// TIA Portal V17 export
// export: Created 2025-03-07T09:24:06.9571705Z, ExportSetting WithDefaults, DisplayName Totally Integrated Automation Portal, DisplayVersion V17 Update 8, DisplayName TIA Portal Openness, DisplayVersion V17 Update 8, DisplayName TIA Portal Version Control Interface, DisplayVersion V17, DisplayName SINAMICS Startdrive Advanced, DisplayVersion V17 SP2, DisplayName SINAMICS Startdrive G110M, G120, G120C, G120D, G120P, G115D, DisplayVersion V17 SP2, DisplayName SINAMICS Startdrive G130, G150, S120, S150, SINAMICS MV, S210, DisplayVersion V17 SP2, DisplayName STEP 7 Professional, DisplayVersion V17 Update 8, DisplayName SINUMERIK ONE STEP 7 Toolbox, DisplayVersion V17 Update 12, DisplayName SINUMERIK 840D sl STEP 7 Toolbox, DisplayVersion V17 Update 12, DisplayName STEP 7 Safety, DisplayVersion V17 Update 6, DisplayName WinCC Advanced, DisplayVersion V17 Update 8
FUNCTION "FC22701_LOAD_FEEDER_SEQUENCES" : Void   // FC22701, LAD
TITLE = FC22701 LOAD FEEDER SEQUENCES
{ S7_Optimized_Access := 'TRUE' }
VERSION : 0.1
// stored: AutoNumber false, IsIECCheckEnabled false, SetENOAutomatically false, UDAEnableTagReadback false
BEGIN

REGION Network 1: //////////_UNIT_01_//////////
END_REGION

REGION Network 2: /////_HOPPER_1_SEQUENCES_/////
END_REGION

REGION Network 3: CALL FB22701 LOAD FEEDER SEQUENCE TIME UNIT 01 HOPPER 1
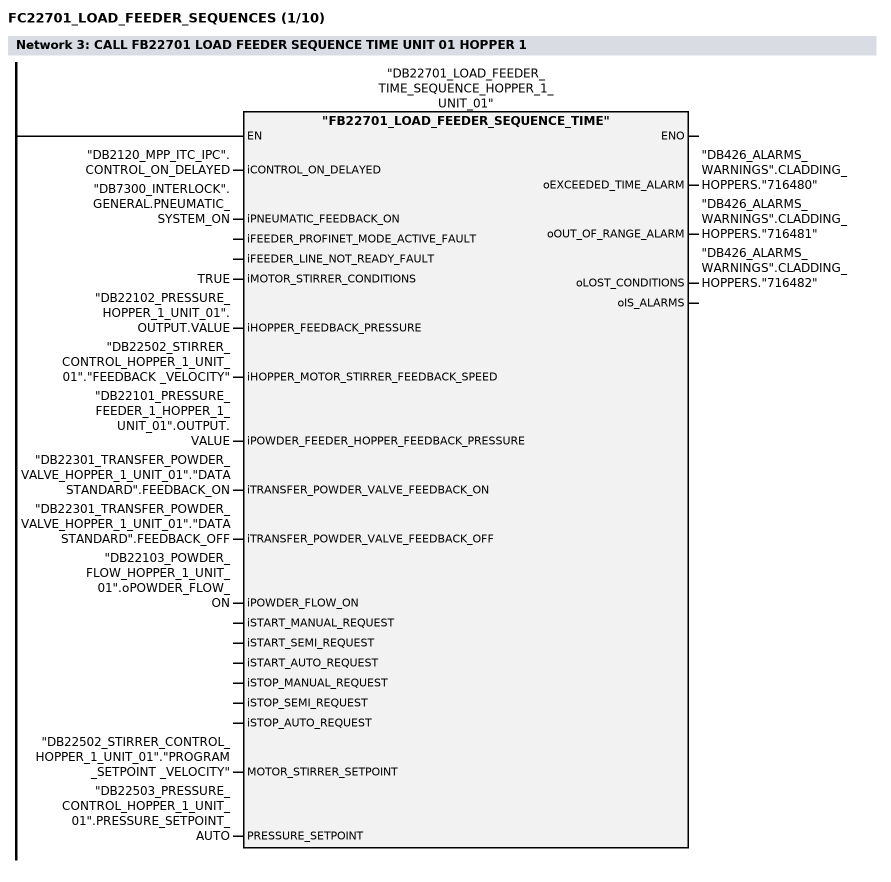
   RUNG wire#powerrail
      "DB22701_LOAD_FEEDER_TIME_SEQUENCE_HOPPER_1_UNIT_01"(iCONTROL_ON_DELAYED := "DB2120_MPP_ITC_IPC".CONTROL_ON_DELAYED, iPNEUMATIC_FEEDBACK_ON := "DB7300_INTERLOCK".GENERAL.PNEUMATIC_SYSTEM_ON, iFEEDER_PROFINET_MODE_ACTIVE_FAULT :=, iFEEDER_LINE_NOT_READY_FAULT :=, iMOTOR_STIRRER_CONDITIONS := TRUE, iHOPPER_FEEDBACK_PRESSURE := "DB22102_PRESSURE_HOPPER_1_UNIT_01".OUTPUT.VALUE, iHOPPER_MOTOR_STIRRER_FEEDBACK_SPEED := "DB22502_STIRRER_CONTROL_HOPPER_1_UNIT_01"."FEEDBACK _VELOCITY", iPOWDER_FEEDER_HOPPER_FEEDBACK_PRESSURE := "DB22101_PRESSURE_FEEDER_1_HOPPER_1_UNIT_01".OUTPUT.VALUE, iTRANSFER_POWDER_VALVE_FEEDBACK_ON := "DB22301_TRANSFER_POWDER_VALVE_HOPPER_1_UNIT_01"."DATA STANDARD".FEEDBACK_ON, iTRANSFER_POWDER_VALVE_FEEDBACK_OFF := "DB22301_TRANSFER_POWDER_VALVE_HOPPER_1_UNIT_01"."DATA STANDARD".FEEDBACK_OFF, iPOWDER_FLOW_ON := "DB22103_POWDER_FLOW_HOPPER_1_UNIT_01".oPOWDER_FLOW_ON, iSTART_MANUAL_REQUEST :=, iSTART_SEMI_REQUEST :=, iSTART_AUTO_REQUEST :=, iSTOP_MANUAL_REQUEST :=, iSTOP_SEMI_REQUEST :=, iSTOP_AUTO_REQUEST :=, MOTOR_STIRRER_SETPOINT := "DB22502_STIRRER_CONTROL_HOPPER_1_UNIT_01"."PROGRAM _SETPOINT _VELOCITY", PRESSURE_SETPOINT := "DB22503_PRESSURE_CONTROL_HOPPER_1_UNIT_01".PRESSURE_SETPOINT_AUTO, oEXCEEDED_TIME_ALARM => "DB426_ALARMS_WARNINGS".CLADDING_HOPPERS."716480", oOUT_OF_RANGE_ALARM => "DB426_ALARMS_WARNINGS".CLADDING_HOPPERS."716481", oLOST_CONDITIONS => "DB426_ALARMS_WARNINGS".CLADDING_HOPPERS."716482", oIS_ALARMS =>)
   END_RUNG
   // the same network as SCL:
   "DB22701_LOAD_FEEDER_TIME_SEQUENCE_HOPPER_1_UNIT_01"(iCONTROL_ON_DELAYED := "DB2120_MPP_ITC_IPC".CONTROL_ON_DELAYED,   // "FB22701_LOAD_FEEDER_SEQUENCE_TIME"
                           iPNEUMATIC_FEEDBACK_ON := "DB7300_INTERLOCK".GENERAL.PNEUMATIC_SYSTEM_ON,
                           iMOTOR_STIRRER_CONDITIONS := TRUE,
                           iHOPPER_FEEDBACK_PRESSURE := "DB22102_PRESSURE_HOPPER_1_UNIT_01".OUTPUT.VALUE,
                           iHOPPER_MOTOR_STIRRER_FEEDBACK_SPEED := "DB22502_STIRRER_CONTROL_HOPPER_1_UNIT_01"."FEEDBACK _VELOCITY",
                           iPOWDER_FEEDER_HOPPER_FEEDBACK_PRESSURE := "DB22101_PRESSURE_FEEDER_1_HOPPER_1_UNIT_01".OUTPUT.VALUE,
                           iTRANSFER_POWDER_VALVE_FEEDBACK_ON := "DB22301_TRANSFER_POWDER_VALVE_HOPPER_1_UNIT_01"."DATA STANDARD".FEEDBACK_ON,
                           iTRANSFER_POWDER_VALVE_FEEDBACK_OFF := "DB22301_TRANSFER_POWDER_VALVE_HOPPER_1_UNIT_01"."DATA STANDARD".FEEDBACK_OFF,
                           iPOWDER_FLOW_ON := "DB22103_POWDER_FLOW_HOPPER_1_UNIT_01".oPOWDER_FLOW_ON,
                           MOTOR_STIRRER_SETPOINT := "DB22502_STIRRER_CONTROL_HOPPER_1_UNIT_01"."PROGRAM _SETPOINT _VELOCITY",
                           PRESSURE_SETPOINT := "DB22503_PRESSURE_CONTROL_HOPPER_1_UNIT_01".PRESSURE_SETPOINT_AUTO,
                           oEXCEEDED_TIME_ALARM => "DB426_ALARMS_WARNINGS".CLADDING_HOPPERS."716480",
                           oOUT_OF_RANGE_ALARM => "DB426_ALARMS_WARNINGS".CLADDING_HOPPERS."716481",
                           oLOST_CONDITIONS => "DB426_ALARMS_WARNINGS".CLADDING_HOPPERS."716482");
END_REGION

REGION Network 4: CALL FB22702 LOAD FEEDER SEQUENCE WEIGHT UNIT 01 HOPPER 1
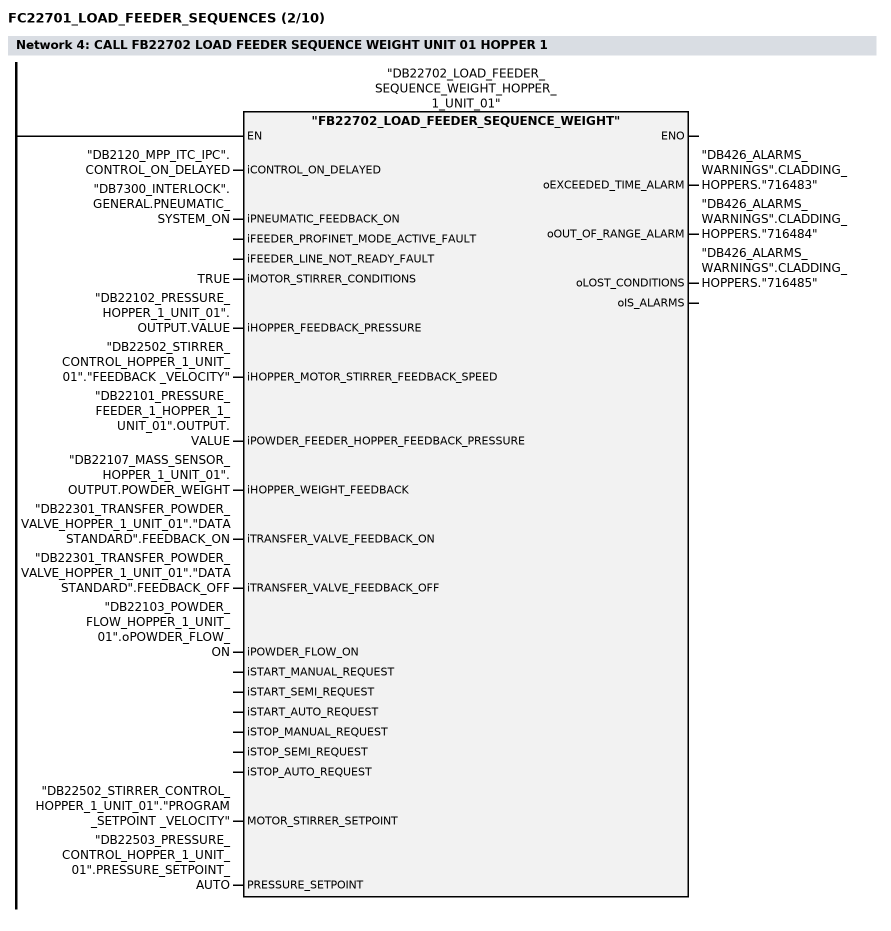
   RUNG wire#powerrail
      "DB22702_LOAD_FEEDER_SEQUENCE_WEIGHT_HOPPER_1_UNIT_01"(iCONTROL_ON_DELAYED := "DB2120_MPP_ITC_IPC".CONTROL_ON_DELAYED, iPNEUMATIC_FEEDBACK_ON := "DB7300_INTERLOCK".GENERAL.PNEUMATIC_SYSTEM_ON, iFEEDER_PROFINET_MODE_ACTIVE_FAULT :=, iFEEDER_LINE_NOT_READY_FAULT :=, iMOTOR_STIRRER_CONDITIONS := TRUE, iHOPPER_FEEDBACK_PRESSURE := "DB22102_PRESSURE_HOPPER_1_UNIT_01".OUTPUT.VALUE, iHOPPER_MOTOR_STIRRER_FEEDBACK_SPEED := "DB22502_STIRRER_CONTROL_HOPPER_1_UNIT_01"."FEEDBACK _VELOCITY", iPOWDER_FEEDER_HOPPER_FEEDBACK_PRESSURE := "DB22101_PRESSURE_FEEDER_1_HOPPER_1_UNIT_01".OUTPUT.VALUE, iHOPPER_WEIGHT_FEEDBACK := "DB22107_MASS_SENSOR_HOPPER_1_UNIT_01".OUTPUT.POWDER_WEIGHT, iTRANSFER_VALVE_FEEDBACK_ON := "DB22301_TRANSFER_POWDER_VALVE_HOPPER_1_UNIT_01"."DATA STANDARD".FEEDBACK_ON, iTRANSFER_VALVE_FEEDBACK_OFF := "DB22301_TRANSFER_POWDER_VALVE_HOPPER_1_UNIT_01"."DATA STANDARD".FEEDBACK_OFF, iPOWDER_FLOW_ON := "DB22103_POWDER_FLOW_HOPPER_1_UNIT_01".oPOWDER_FLOW_ON, iSTART_MANUAL_REQUEST :=, iSTART_SEMI_REQUEST :=, iSTART_AUTO_REQUEST :=, iSTOP_MANUAL_REQUEST :=, iSTOP_SEMI_REQUEST :=, iSTOP_AUTO_REQUEST :=, MOTOR_STIRRER_SETPOINT := "DB22502_STIRRER_CONTROL_HOPPER_1_UNIT_01"."PROGRAM _SETPOINT _VELOCITY", PRESSURE_SETPOINT := "DB22503_PRESSURE_CONTROL_HOPPER_1_UNIT_01".PRESSURE_SETPOINT_AUTO, oEXCEEDED_TIME_ALARM => "DB426_ALARMS_WARNINGS".CLADDING_HOPPERS."716483", oOUT_OF_RANGE_ALARM => "DB426_ALARMS_WARNINGS".CLADDING_HOPPERS."716484", oLOST_CONDITIONS => "DB426_ALARMS_WARNINGS".CLADDING_HOPPERS."716485", oIS_ALARMS =>)
   END_RUNG
   // the same network as SCL:
   "DB22702_LOAD_FEEDER_SEQUENCE_WEIGHT_HOPPER_1_UNIT_01"(iCONTROL_ON_DELAYED := "DB2120_MPP_ITC_IPC".CONTROL_ON_DELAYED,   // "FB22702_LOAD_FEEDER_SEQUENCE_WEIGHT"
                           iPNEUMATIC_FEEDBACK_ON := "DB7300_INTERLOCK".GENERAL.PNEUMATIC_SYSTEM_ON,
                           iMOTOR_STIRRER_CONDITIONS := TRUE,
                           iHOPPER_FEEDBACK_PRESSURE := "DB22102_PRESSURE_HOPPER_1_UNIT_01".OUTPUT.VALUE,
                           iHOPPER_MOTOR_STIRRER_FEEDBACK_SPEED := "DB22502_STIRRER_CONTROL_HOPPER_1_UNIT_01"."FEEDBACK _VELOCITY",
                           iPOWDER_FEEDER_HOPPER_FEEDBACK_PRESSURE := "DB22101_PRESSURE_FEEDER_1_HOPPER_1_UNIT_01".OUTPUT.VALUE,
                           iHOPPER_WEIGHT_FEEDBACK := "DB22107_MASS_SENSOR_HOPPER_1_UNIT_01".OUTPUT.POWDER_WEIGHT,
                           iTRANSFER_VALVE_FEEDBACK_ON := "DB22301_TRANSFER_POWDER_VALVE_HOPPER_1_UNIT_01"."DATA STANDARD".FEEDBACK_ON,
                           iTRANSFER_VALVE_FEEDBACK_OFF := "DB22301_TRANSFER_POWDER_VALVE_HOPPER_1_UNIT_01"."DATA STANDARD".FEEDBACK_OFF,
                           iPOWDER_FLOW_ON := "DB22103_POWDER_FLOW_HOPPER_1_UNIT_01".oPOWDER_FLOW_ON,
                           MOTOR_STIRRER_SETPOINT := "DB22502_STIRRER_CONTROL_HOPPER_1_UNIT_01"."PROGRAM _SETPOINT _VELOCITY",
                           PRESSURE_SETPOINT := "DB22503_PRESSURE_CONTROL_HOPPER_1_UNIT_01".PRESSURE_SETPOINT_AUTO,
                           oEXCEEDED_TIME_ALARM => "DB426_ALARMS_WARNINGS".CLADDING_HOPPERS."716483",
                           oOUT_OF_RANGE_ALARM => "DB426_ALARMS_WARNINGS".CLADDING_HOPPERS."716484",
                           oLOST_CONDITIONS => "DB426_ALARMS_WARNINGS".CLADDING_HOPPERS."716485");
END_REGION

REGION Network 5: /////_HOPPER_2_SEQUENCES_/////
END_REGION

REGION Network 6: CALL FB22701 LOAD FEEDER SEQUENCE TIME UNIT 01 HOPPER 2
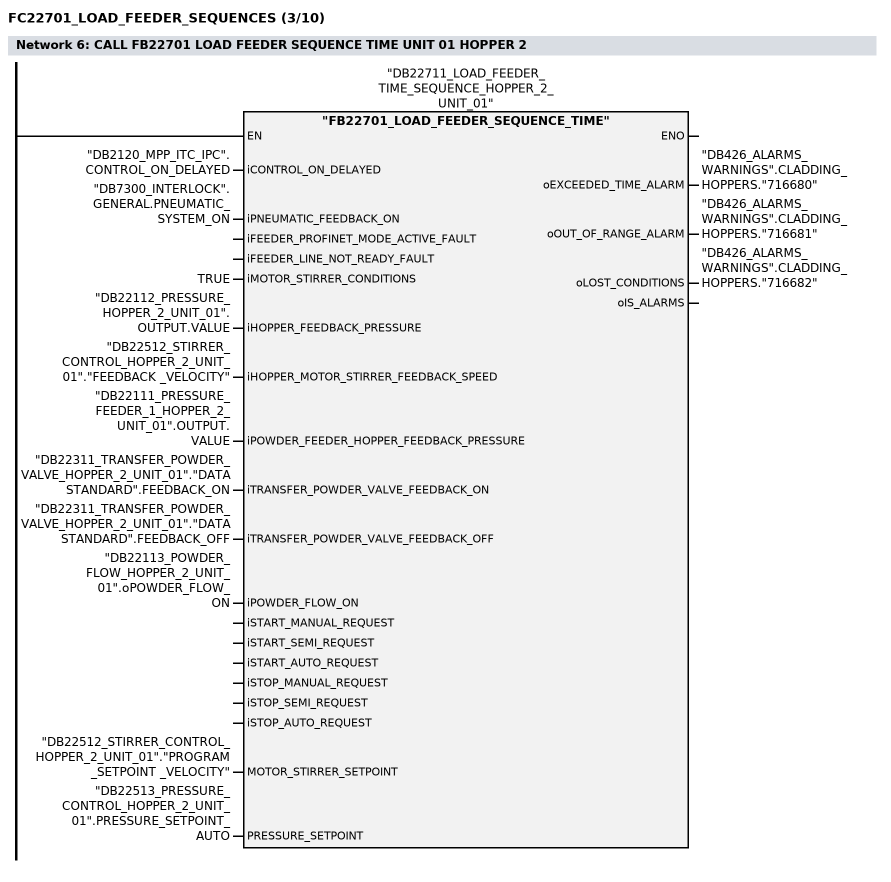
   RUNG wire#powerrail
      "DB22711_LOAD_FEEDER_TIME_SEQUENCE_HOPPER_2_UNIT_01"(iCONTROL_ON_DELAYED := "DB2120_MPP_ITC_IPC".CONTROL_ON_DELAYED, iPNEUMATIC_FEEDBACK_ON := "DB7300_INTERLOCK".GENERAL.PNEUMATIC_SYSTEM_ON, iFEEDER_PROFINET_MODE_ACTIVE_FAULT :=, iFEEDER_LINE_NOT_READY_FAULT :=, iMOTOR_STIRRER_CONDITIONS := TRUE, iHOPPER_FEEDBACK_PRESSURE := "DB22112_PRESSURE_HOPPER_2_UNIT_01".OUTPUT.VALUE, iHOPPER_MOTOR_STIRRER_FEEDBACK_SPEED := "DB22512_STIRRER_CONTROL_HOPPER_2_UNIT_01"."FEEDBACK _VELOCITY", iPOWDER_FEEDER_HOPPER_FEEDBACK_PRESSURE := "DB22111_PRESSURE_FEEDER_1_HOPPER_2_UNIT_01".OUTPUT.VALUE, iTRANSFER_POWDER_VALVE_FEEDBACK_ON := "DB22311_TRANSFER_POWDER_VALVE_HOPPER_2_UNIT_01"."DATA STANDARD".FEEDBACK_ON, iTRANSFER_POWDER_VALVE_FEEDBACK_OFF := "DB22311_TRANSFER_POWDER_VALVE_HOPPER_2_UNIT_01"."DATA STANDARD".FEEDBACK_OFF, iPOWDER_FLOW_ON := "DB22113_POWDER_FLOW_HOPPER_2_UNIT_01".oPOWDER_FLOW_ON, iSTART_MANUAL_REQUEST :=, iSTART_SEMI_REQUEST :=, iSTART_AUTO_REQUEST :=, iSTOP_MANUAL_REQUEST :=, iSTOP_SEMI_REQUEST :=, iSTOP_AUTO_REQUEST :=, MOTOR_STIRRER_SETPOINT := "DB22512_STIRRER_CONTROL_HOPPER_2_UNIT_01"."PROGRAM _SETPOINT _VELOCITY", PRESSURE_SETPOINT := "DB22513_PRESSURE_CONTROL_HOPPER_2_UNIT_01".PRESSURE_SETPOINT_AUTO, oEXCEEDED_TIME_ALARM => "DB426_ALARMS_WARNINGS".CLADDING_HOPPERS."716680", oOUT_OF_RANGE_ALARM => "DB426_ALARMS_WARNINGS".CLADDING_HOPPERS."716681", oLOST_CONDITIONS => "DB426_ALARMS_WARNINGS".CLADDING_HOPPERS."716682", oIS_ALARMS =>)
   END_RUNG
   // the same network as SCL:
   "DB22711_LOAD_FEEDER_TIME_SEQUENCE_HOPPER_2_UNIT_01"(iCONTROL_ON_DELAYED := "DB2120_MPP_ITC_IPC".CONTROL_ON_DELAYED,   // "FB22701_LOAD_FEEDER_SEQUENCE_TIME"
                           iPNEUMATIC_FEEDBACK_ON := "DB7300_INTERLOCK".GENERAL.PNEUMATIC_SYSTEM_ON,
                           iMOTOR_STIRRER_CONDITIONS := TRUE,
                           iHOPPER_FEEDBACK_PRESSURE := "DB22112_PRESSURE_HOPPER_2_UNIT_01".OUTPUT.VALUE,
                           iHOPPER_MOTOR_STIRRER_FEEDBACK_SPEED := "DB22512_STIRRER_CONTROL_HOPPER_2_UNIT_01"."FEEDBACK _VELOCITY",
                           iPOWDER_FEEDER_HOPPER_FEEDBACK_PRESSURE := "DB22111_PRESSURE_FEEDER_1_HOPPER_2_UNIT_01".OUTPUT.VALUE,
                           iTRANSFER_POWDER_VALVE_FEEDBACK_ON := "DB22311_TRANSFER_POWDER_VALVE_HOPPER_2_UNIT_01"."DATA STANDARD".FEEDBACK_ON,
                           iTRANSFER_POWDER_VALVE_FEEDBACK_OFF := "DB22311_TRANSFER_POWDER_VALVE_HOPPER_2_UNIT_01"."DATA STANDARD".FEEDBACK_OFF,
                           iPOWDER_FLOW_ON := "DB22113_POWDER_FLOW_HOPPER_2_UNIT_01".oPOWDER_FLOW_ON,
                           MOTOR_STIRRER_SETPOINT := "DB22512_STIRRER_CONTROL_HOPPER_2_UNIT_01"."PROGRAM _SETPOINT _VELOCITY",
                           PRESSURE_SETPOINT := "DB22513_PRESSURE_CONTROL_HOPPER_2_UNIT_01".PRESSURE_SETPOINT_AUTO,
                           oEXCEEDED_TIME_ALARM => "DB426_ALARMS_WARNINGS".CLADDING_HOPPERS."716680",
                           oOUT_OF_RANGE_ALARM => "DB426_ALARMS_WARNINGS".CLADDING_HOPPERS."716681",
                           oLOST_CONDITIONS => "DB426_ALARMS_WARNINGS".CLADDING_HOPPERS."716682");
END_REGION

REGION Network 7: CALL FB22702 LOAD FEEDER SEQUENCE WEIGHT UNIT 01 HOPPER 2
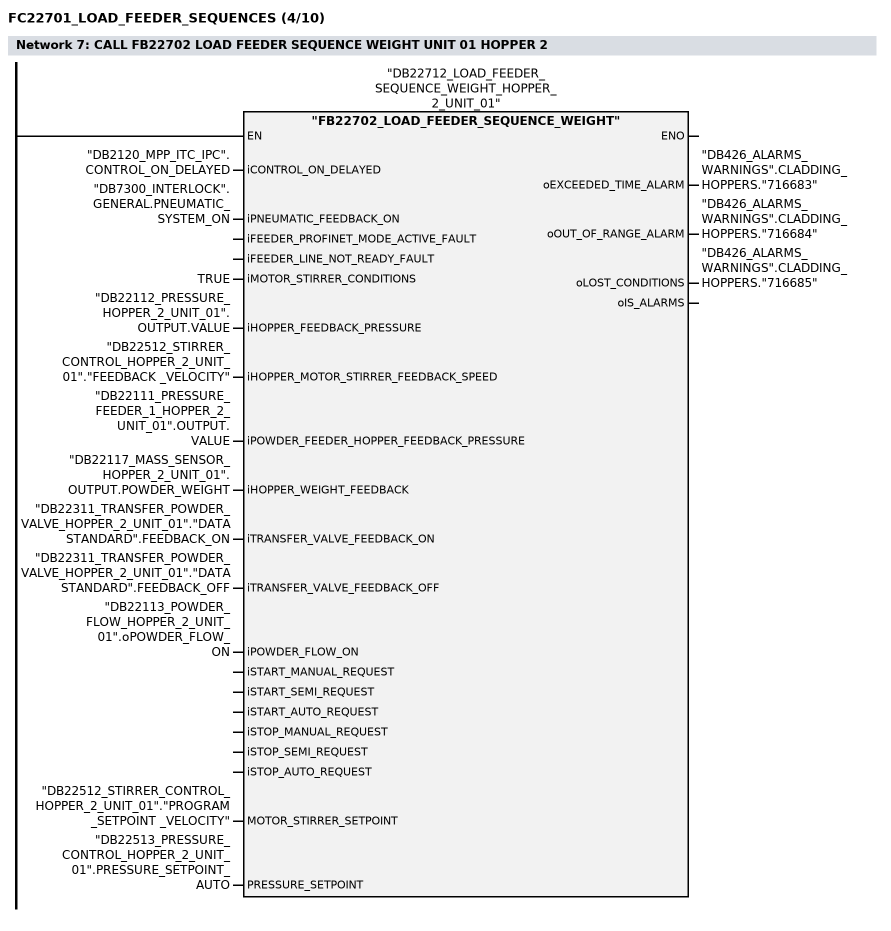
   RUNG wire#powerrail
      "DB22712_LOAD_FEEDER_SEQUENCE_WEIGHT_HOPPER_2_UNIT_01"(iCONTROL_ON_DELAYED := "DB2120_MPP_ITC_IPC".CONTROL_ON_DELAYED, iPNEUMATIC_FEEDBACK_ON := "DB7300_INTERLOCK".GENERAL.PNEUMATIC_SYSTEM_ON, iFEEDER_PROFINET_MODE_ACTIVE_FAULT :=, iFEEDER_LINE_NOT_READY_FAULT :=, iMOTOR_STIRRER_CONDITIONS := TRUE, iHOPPER_FEEDBACK_PRESSURE := "DB22112_PRESSURE_HOPPER_2_UNIT_01".OUTPUT.VALUE, iHOPPER_MOTOR_STIRRER_FEEDBACK_SPEED := "DB22512_STIRRER_CONTROL_HOPPER_2_UNIT_01"."FEEDBACK _VELOCITY", iPOWDER_FEEDER_HOPPER_FEEDBACK_PRESSURE := "DB22111_PRESSURE_FEEDER_1_HOPPER_2_UNIT_01".OUTPUT.VALUE, iHOPPER_WEIGHT_FEEDBACK := "DB22117_MASS_SENSOR_HOPPER_2_UNIT_01".OUTPUT.POWDER_WEIGHT, iTRANSFER_VALVE_FEEDBACK_ON := "DB22311_TRANSFER_POWDER_VALVE_HOPPER_2_UNIT_01"."DATA STANDARD".FEEDBACK_ON, iTRANSFER_VALVE_FEEDBACK_OFF := "DB22311_TRANSFER_POWDER_VALVE_HOPPER_2_UNIT_01"."DATA STANDARD".FEEDBACK_OFF, iPOWDER_FLOW_ON := "DB22113_POWDER_FLOW_HOPPER_2_UNIT_01".oPOWDER_FLOW_ON, iSTART_MANUAL_REQUEST :=, iSTART_SEMI_REQUEST :=, iSTART_AUTO_REQUEST :=, iSTOP_MANUAL_REQUEST :=, iSTOP_SEMI_REQUEST :=, iSTOP_AUTO_REQUEST :=, MOTOR_STIRRER_SETPOINT := "DB22512_STIRRER_CONTROL_HOPPER_2_UNIT_01"."PROGRAM _SETPOINT _VELOCITY", PRESSURE_SETPOINT := "DB22513_PRESSURE_CONTROL_HOPPER_2_UNIT_01".PRESSURE_SETPOINT_AUTO, oEXCEEDED_TIME_ALARM => "DB426_ALARMS_WARNINGS".CLADDING_HOPPERS."716683", oOUT_OF_RANGE_ALARM => "DB426_ALARMS_WARNINGS".CLADDING_HOPPERS."716684", oLOST_CONDITIONS => "DB426_ALARMS_WARNINGS".CLADDING_HOPPERS."716685", oIS_ALARMS =>)
   END_RUNG
   // the same network as SCL:
   "DB22712_LOAD_FEEDER_SEQUENCE_WEIGHT_HOPPER_2_UNIT_01"(iCONTROL_ON_DELAYED := "DB2120_MPP_ITC_IPC".CONTROL_ON_DELAYED,   // "FB22702_LOAD_FEEDER_SEQUENCE_WEIGHT"
                           iPNEUMATIC_FEEDBACK_ON := "DB7300_INTERLOCK".GENERAL.PNEUMATIC_SYSTEM_ON,
                           iMOTOR_STIRRER_CONDITIONS := TRUE,
                           iHOPPER_FEEDBACK_PRESSURE := "DB22112_PRESSURE_HOPPER_2_UNIT_01".OUTPUT.VALUE,
                           iHOPPER_MOTOR_STIRRER_FEEDBACK_SPEED := "DB22512_STIRRER_CONTROL_HOPPER_2_UNIT_01"."FEEDBACK _VELOCITY",
                           iPOWDER_FEEDER_HOPPER_FEEDBACK_PRESSURE := "DB22111_PRESSURE_FEEDER_1_HOPPER_2_UNIT_01".OUTPUT.VALUE,
                           iHOPPER_WEIGHT_FEEDBACK := "DB22117_MASS_SENSOR_HOPPER_2_UNIT_01".OUTPUT.POWDER_WEIGHT,
                           iTRANSFER_VALVE_FEEDBACK_ON := "DB22311_TRANSFER_POWDER_VALVE_HOPPER_2_UNIT_01"."DATA STANDARD".FEEDBACK_ON,
                           iTRANSFER_VALVE_FEEDBACK_OFF := "DB22311_TRANSFER_POWDER_VALVE_HOPPER_2_UNIT_01"."DATA STANDARD".FEEDBACK_OFF,
                           iPOWDER_FLOW_ON := "DB22113_POWDER_FLOW_HOPPER_2_UNIT_01".oPOWDER_FLOW_ON,
                           MOTOR_STIRRER_SETPOINT := "DB22512_STIRRER_CONTROL_HOPPER_2_UNIT_01"."PROGRAM _SETPOINT _VELOCITY",
                           PRESSURE_SETPOINT := "DB22513_PRESSURE_CONTROL_HOPPER_2_UNIT_01".PRESSURE_SETPOINT_AUTO,
                           oEXCEEDED_TIME_ALARM => "DB426_ALARMS_WARNINGS".CLADDING_HOPPERS."716683",
                           oOUT_OF_RANGE_ALARM => "DB426_ALARMS_WARNINGS".CLADDING_HOPPERS."716684",
                           oLOST_CONDITIONS => "DB426_ALARMS_WARNINGS".CLADDING_HOPPERS."716685");
END_REGION

REGION Network 8: //////////_UNIT_02_//////////
END_REGION

REGION Network 9: /////_HOPPER_1_SEQUENCES_/////
END_REGION

REGION Network 10: CALL FB22701 LOAD FEEDER SEQUENCE TIME UNIT 02 HOPPER 1
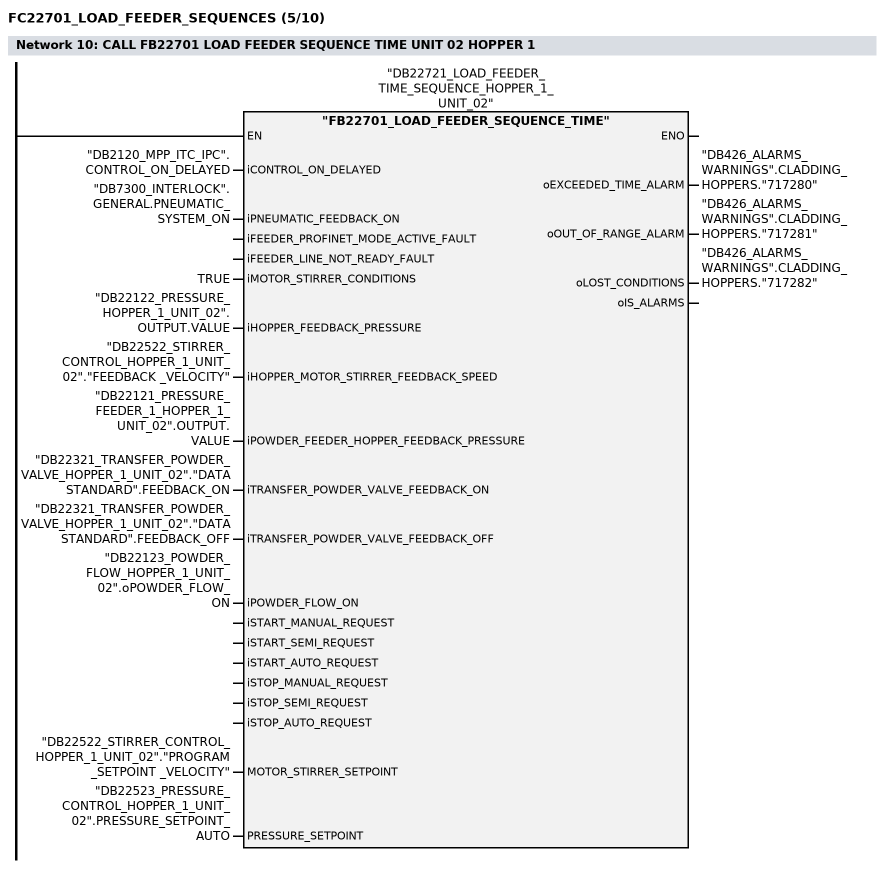
   RUNG wire#powerrail
      "DB22721_LOAD_FEEDER_TIME_SEQUENCE_HOPPER_1_UNIT_02"(iCONTROL_ON_DELAYED := "DB2120_MPP_ITC_IPC".CONTROL_ON_DELAYED, iPNEUMATIC_FEEDBACK_ON := "DB7300_INTERLOCK".GENERAL.PNEUMATIC_SYSTEM_ON, iFEEDER_PROFINET_MODE_ACTIVE_FAULT :=, iFEEDER_LINE_NOT_READY_FAULT :=, iMOTOR_STIRRER_CONDITIONS := TRUE, iHOPPER_FEEDBACK_PRESSURE := "DB22122_PRESSURE_HOPPER_1_UNIT_02".OUTPUT.VALUE, iHOPPER_MOTOR_STIRRER_FEEDBACK_SPEED := "DB22522_STIRRER_CONTROL_HOPPER_1_UNIT_02"."FEEDBACK _VELOCITY", iPOWDER_FEEDER_HOPPER_FEEDBACK_PRESSURE := "DB22121_PRESSURE_FEEDER_1_HOPPER_1_UNIT_02".OUTPUT.VALUE, iTRANSFER_POWDER_VALVE_FEEDBACK_ON := "DB22321_TRANSFER_POWDER_VALVE_HOPPER_1_UNIT_02"."DATA STANDARD".FEEDBACK_ON, iTRANSFER_POWDER_VALVE_FEEDBACK_OFF := "DB22321_TRANSFER_POWDER_VALVE_HOPPER_1_UNIT_02"."DATA STANDARD".FEEDBACK_OFF, iPOWDER_FLOW_ON := "DB22123_POWDER_FLOW_HOPPER_1_UNIT_02".oPOWDER_FLOW_ON, iSTART_MANUAL_REQUEST :=, iSTART_SEMI_REQUEST :=, iSTART_AUTO_REQUEST :=, iSTOP_MANUAL_REQUEST :=, iSTOP_SEMI_REQUEST :=, iSTOP_AUTO_REQUEST :=, MOTOR_STIRRER_SETPOINT := "DB22522_STIRRER_CONTROL_HOPPER_1_UNIT_02"."PROGRAM _SETPOINT _VELOCITY", PRESSURE_SETPOINT := "DB22523_PRESSURE_CONTROL_HOPPER_1_UNIT_02".PRESSURE_SETPOINT_AUTO, oEXCEEDED_TIME_ALARM => "DB426_ALARMS_WARNINGS".CLADDING_HOPPERS."717280", oOUT_OF_RANGE_ALARM => "DB426_ALARMS_WARNINGS".CLADDING_HOPPERS."717281", oLOST_CONDITIONS => "DB426_ALARMS_WARNINGS".CLADDING_HOPPERS."717282", oIS_ALARMS =>)
   END_RUNG
   // the same network as SCL:
   "DB22721_LOAD_FEEDER_TIME_SEQUENCE_HOPPER_1_UNIT_02"(iCONTROL_ON_DELAYED := "DB2120_MPP_ITC_IPC".CONTROL_ON_DELAYED,   // "FB22701_LOAD_FEEDER_SEQUENCE_TIME"
                           iPNEUMATIC_FEEDBACK_ON := "DB7300_INTERLOCK".GENERAL.PNEUMATIC_SYSTEM_ON,
                           iMOTOR_STIRRER_CONDITIONS := TRUE,
                           iHOPPER_FEEDBACK_PRESSURE := "DB22122_PRESSURE_HOPPER_1_UNIT_02".OUTPUT.VALUE,
                           iHOPPER_MOTOR_STIRRER_FEEDBACK_SPEED := "DB22522_STIRRER_CONTROL_HOPPER_1_UNIT_02"."FEEDBACK _VELOCITY",
                           iPOWDER_FEEDER_HOPPER_FEEDBACK_PRESSURE := "DB22121_PRESSURE_FEEDER_1_HOPPER_1_UNIT_02".OUTPUT.VALUE,
                           iTRANSFER_POWDER_VALVE_FEEDBACK_ON := "DB22321_TRANSFER_POWDER_VALVE_HOPPER_1_UNIT_02"."DATA STANDARD".FEEDBACK_ON,
                           iTRANSFER_POWDER_VALVE_FEEDBACK_OFF := "DB22321_TRANSFER_POWDER_VALVE_HOPPER_1_UNIT_02"."DATA STANDARD".FEEDBACK_OFF,
                           iPOWDER_FLOW_ON := "DB22123_POWDER_FLOW_HOPPER_1_UNIT_02".oPOWDER_FLOW_ON,
                           MOTOR_STIRRER_SETPOINT := "DB22522_STIRRER_CONTROL_HOPPER_1_UNIT_02"."PROGRAM _SETPOINT _VELOCITY",
                           PRESSURE_SETPOINT := "DB22523_PRESSURE_CONTROL_HOPPER_1_UNIT_02".PRESSURE_SETPOINT_AUTO,
                           oEXCEEDED_TIME_ALARM => "DB426_ALARMS_WARNINGS".CLADDING_HOPPERS."717280",
                           oOUT_OF_RANGE_ALARM => "DB426_ALARMS_WARNINGS".CLADDING_HOPPERS."717281",
                           oLOST_CONDITIONS => "DB426_ALARMS_WARNINGS".CLADDING_HOPPERS."717282");
END_REGION

REGION Network 11: CALL FB22702 LOAD FEEDER SEQUENCE WEIGHT UNIT 02 HOPPER 1
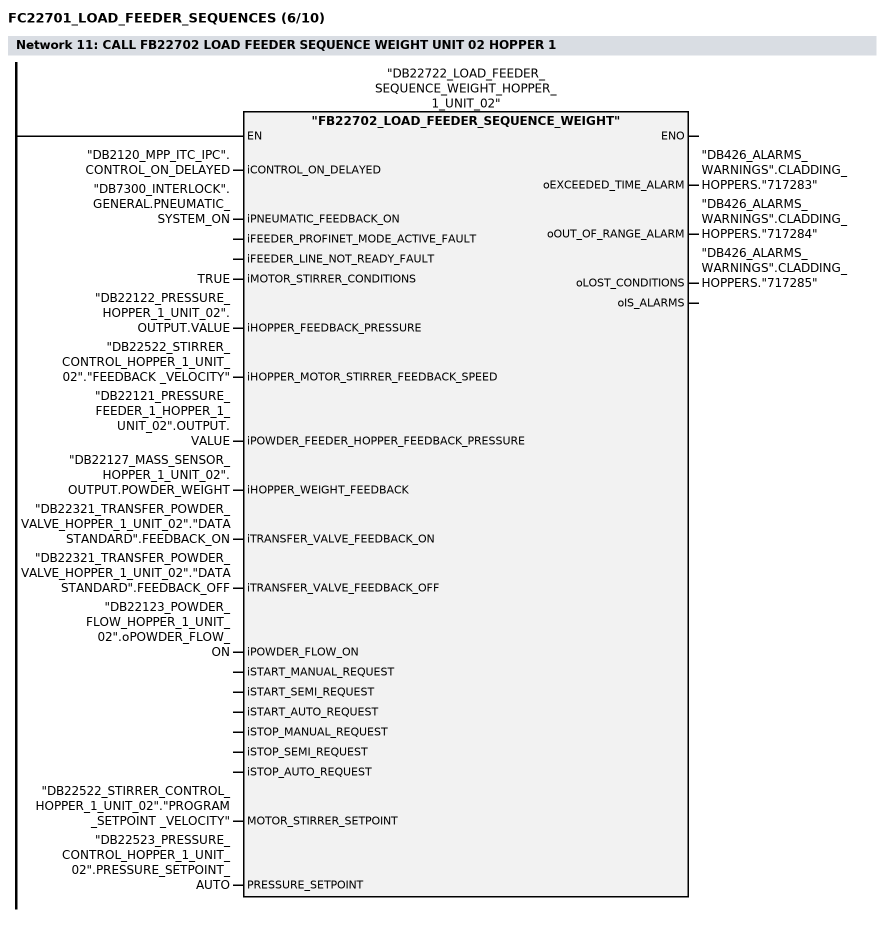
   RUNG wire#powerrail
      "DB22722_LOAD_FEEDER_SEQUENCE_WEIGHT_HOPPER_1_UNIT_02"(iCONTROL_ON_DELAYED := "DB2120_MPP_ITC_IPC".CONTROL_ON_DELAYED, iPNEUMATIC_FEEDBACK_ON := "DB7300_INTERLOCK".GENERAL.PNEUMATIC_SYSTEM_ON, iFEEDER_PROFINET_MODE_ACTIVE_FAULT :=, iFEEDER_LINE_NOT_READY_FAULT :=, iMOTOR_STIRRER_CONDITIONS := TRUE, iHOPPER_FEEDBACK_PRESSURE := "DB22122_PRESSURE_HOPPER_1_UNIT_02".OUTPUT.VALUE, iHOPPER_MOTOR_STIRRER_FEEDBACK_SPEED := "DB22522_STIRRER_CONTROL_HOPPER_1_UNIT_02"."FEEDBACK _VELOCITY", iPOWDER_FEEDER_HOPPER_FEEDBACK_PRESSURE := "DB22121_PRESSURE_FEEDER_1_HOPPER_1_UNIT_02".OUTPUT.VALUE, iHOPPER_WEIGHT_FEEDBACK := "DB22127_MASS_SENSOR_HOPPER_1_UNIT_02".OUTPUT.POWDER_WEIGHT, iTRANSFER_VALVE_FEEDBACK_ON := "DB22321_TRANSFER_POWDER_VALVE_HOPPER_1_UNIT_02"."DATA STANDARD".FEEDBACK_ON, iTRANSFER_VALVE_FEEDBACK_OFF := "DB22321_TRANSFER_POWDER_VALVE_HOPPER_1_UNIT_02"."DATA STANDARD".FEEDBACK_OFF, iPOWDER_FLOW_ON := "DB22123_POWDER_FLOW_HOPPER_1_UNIT_02".oPOWDER_FLOW_ON, iSTART_MANUAL_REQUEST :=, iSTART_SEMI_REQUEST :=, iSTART_AUTO_REQUEST :=, iSTOP_MANUAL_REQUEST :=, iSTOP_SEMI_REQUEST :=, iSTOP_AUTO_REQUEST :=, MOTOR_STIRRER_SETPOINT := "DB22522_STIRRER_CONTROL_HOPPER_1_UNIT_02"."PROGRAM _SETPOINT _VELOCITY", PRESSURE_SETPOINT := "DB22523_PRESSURE_CONTROL_HOPPER_1_UNIT_02".PRESSURE_SETPOINT_AUTO, oEXCEEDED_TIME_ALARM => "DB426_ALARMS_WARNINGS".CLADDING_HOPPERS."717283", oOUT_OF_RANGE_ALARM => "DB426_ALARMS_WARNINGS".CLADDING_HOPPERS."717284", oLOST_CONDITIONS => "DB426_ALARMS_WARNINGS".CLADDING_HOPPERS."717285", oIS_ALARMS =>)
   END_RUNG
   // the same network as SCL:
   "DB22722_LOAD_FEEDER_SEQUENCE_WEIGHT_HOPPER_1_UNIT_02"(iCONTROL_ON_DELAYED := "DB2120_MPP_ITC_IPC".CONTROL_ON_DELAYED,   // "FB22702_LOAD_FEEDER_SEQUENCE_WEIGHT"
                           iPNEUMATIC_FEEDBACK_ON := "DB7300_INTERLOCK".GENERAL.PNEUMATIC_SYSTEM_ON,
                           iMOTOR_STIRRER_CONDITIONS := TRUE,
                           iHOPPER_FEEDBACK_PRESSURE := "DB22122_PRESSURE_HOPPER_1_UNIT_02".OUTPUT.VALUE,
                           iHOPPER_MOTOR_STIRRER_FEEDBACK_SPEED := "DB22522_STIRRER_CONTROL_HOPPER_1_UNIT_02"."FEEDBACK _VELOCITY",
                           iPOWDER_FEEDER_HOPPER_FEEDBACK_PRESSURE := "DB22121_PRESSURE_FEEDER_1_HOPPER_1_UNIT_02".OUTPUT.VALUE,
                           iHOPPER_WEIGHT_FEEDBACK := "DB22127_MASS_SENSOR_HOPPER_1_UNIT_02".OUTPUT.POWDER_WEIGHT,
                           iTRANSFER_VALVE_FEEDBACK_ON := "DB22321_TRANSFER_POWDER_VALVE_HOPPER_1_UNIT_02"."DATA STANDARD".FEEDBACK_ON,
                           iTRANSFER_VALVE_FEEDBACK_OFF := "DB22321_TRANSFER_POWDER_VALVE_HOPPER_1_UNIT_02"."DATA STANDARD".FEEDBACK_OFF,
                           iPOWDER_FLOW_ON := "DB22123_POWDER_FLOW_HOPPER_1_UNIT_02".oPOWDER_FLOW_ON,
                           MOTOR_STIRRER_SETPOINT := "DB22522_STIRRER_CONTROL_HOPPER_1_UNIT_02"."PROGRAM _SETPOINT _VELOCITY",
                           PRESSURE_SETPOINT := "DB22523_PRESSURE_CONTROL_HOPPER_1_UNIT_02".PRESSURE_SETPOINT_AUTO,
                           oEXCEEDED_TIME_ALARM => "DB426_ALARMS_WARNINGS".CLADDING_HOPPERS."717283",
                           oOUT_OF_RANGE_ALARM => "DB426_ALARMS_WARNINGS".CLADDING_HOPPERS."717284",
                           oLOST_CONDITIONS => "DB426_ALARMS_WARNINGS".CLADDING_HOPPERS."717285");
END_REGION

REGION Network 12: /////_HOPPER_2_SEQUENCES_/////
END_REGION

REGION Network 13: CALL FB22701 LOAD FEEDER SEQUENCE TIME UNIT 02 HOPPER 2
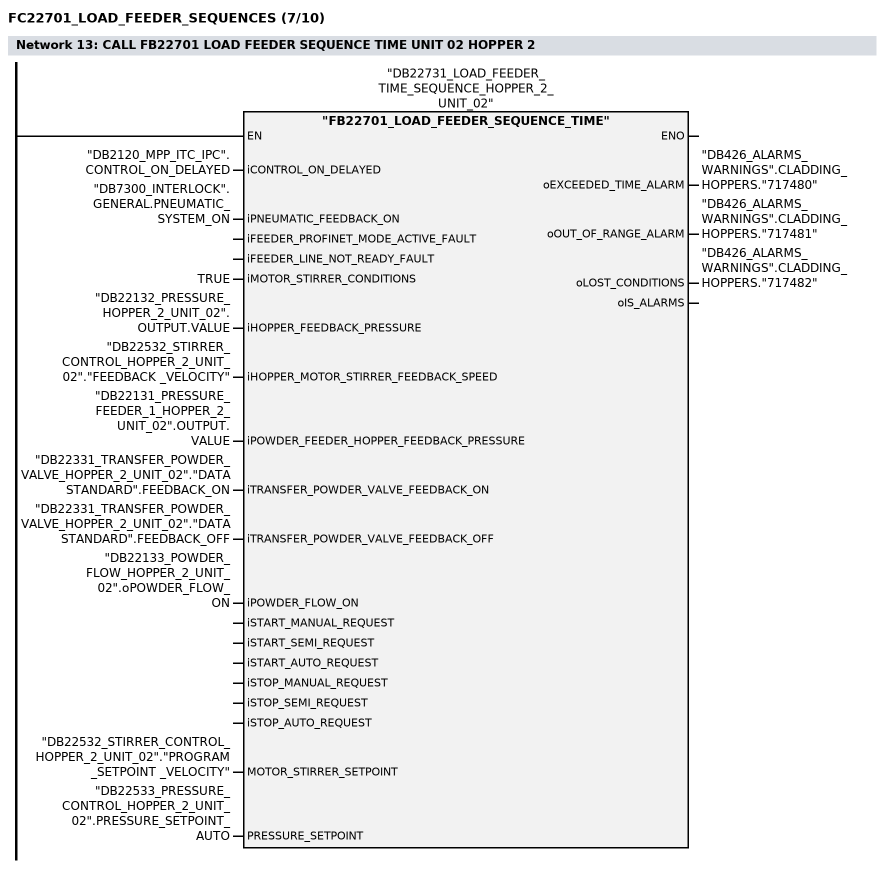
   RUNG wire#powerrail
      "DB22731_LOAD_FEEDER_TIME_SEQUENCE_HOPPER_2_UNIT_02"(iCONTROL_ON_DELAYED := "DB2120_MPP_ITC_IPC".CONTROL_ON_DELAYED, iPNEUMATIC_FEEDBACK_ON := "DB7300_INTERLOCK".GENERAL.PNEUMATIC_SYSTEM_ON, iFEEDER_PROFINET_MODE_ACTIVE_FAULT :=, iFEEDER_LINE_NOT_READY_FAULT :=, iMOTOR_STIRRER_CONDITIONS := TRUE, iHOPPER_FEEDBACK_PRESSURE := "DB22132_PRESSURE_HOPPER_2_UNIT_02".OUTPUT.VALUE, iHOPPER_MOTOR_STIRRER_FEEDBACK_SPEED := "DB22532_STIRRER_CONTROL_HOPPER_2_UNIT_02"."FEEDBACK _VELOCITY", iPOWDER_FEEDER_HOPPER_FEEDBACK_PRESSURE := "DB22131_PRESSURE_FEEDER_1_HOPPER_2_UNIT_02".OUTPUT.VALUE, iTRANSFER_POWDER_VALVE_FEEDBACK_ON := "DB22331_TRANSFER_POWDER_VALVE_HOPPER_2_UNIT_02"."DATA STANDARD".FEEDBACK_ON, iTRANSFER_POWDER_VALVE_FEEDBACK_OFF := "DB22331_TRANSFER_POWDER_VALVE_HOPPER_2_UNIT_02"."DATA STANDARD".FEEDBACK_OFF, iPOWDER_FLOW_ON := "DB22133_POWDER_FLOW_HOPPER_2_UNIT_02".oPOWDER_FLOW_ON, iSTART_MANUAL_REQUEST :=, iSTART_SEMI_REQUEST :=, iSTART_AUTO_REQUEST :=, iSTOP_MANUAL_REQUEST :=, iSTOP_SEMI_REQUEST :=, iSTOP_AUTO_REQUEST :=, MOTOR_STIRRER_SETPOINT := "DB22532_STIRRER_CONTROL_HOPPER_2_UNIT_02"."PROGRAM _SETPOINT _VELOCITY", PRESSURE_SETPOINT := "DB22533_PRESSURE_CONTROL_HOPPER_2_UNIT_02".PRESSURE_SETPOINT_AUTO, oEXCEEDED_TIME_ALARM => "DB426_ALARMS_WARNINGS".CLADDING_HOPPERS."717480", oOUT_OF_RANGE_ALARM => "DB426_ALARMS_WARNINGS".CLADDING_HOPPERS."717481", oLOST_CONDITIONS => "DB426_ALARMS_WARNINGS".CLADDING_HOPPERS."717482", oIS_ALARMS =>)
   END_RUNG
   // the same network as SCL:
   "DB22731_LOAD_FEEDER_TIME_SEQUENCE_HOPPER_2_UNIT_02"(iCONTROL_ON_DELAYED := "DB2120_MPP_ITC_IPC".CONTROL_ON_DELAYED,   // "FB22701_LOAD_FEEDER_SEQUENCE_TIME"
                           iPNEUMATIC_FEEDBACK_ON := "DB7300_INTERLOCK".GENERAL.PNEUMATIC_SYSTEM_ON,
                           iMOTOR_STIRRER_CONDITIONS := TRUE,
                           iHOPPER_FEEDBACK_PRESSURE := "DB22132_PRESSURE_HOPPER_2_UNIT_02".OUTPUT.VALUE,
                           iHOPPER_MOTOR_STIRRER_FEEDBACK_SPEED := "DB22532_STIRRER_CONTROL_HOPPER_2_UNIT_02"."FEEDBACK _VELOCITY",
                           iPOWDER_FEEDER_HOPPER_FEEDBACK_PRESSURE := "DB22131_PRESSURE_FEEDER_1_HOPPER_2_UNIT_02".OUTPUT.VALUE,
                           iTRANSFER_POWDER_VALVE_FEEDBACK_ON := "DB22331_TRANSFER_POWDER_VALVE_HOPPER_2_UNIT_02"."DATA STANDARD".FEEDBACK_ON,
                           iTRANSFER_POWDER_VALVE_FEEDBACK_OFF := "DB22331_TRANSFER_POWDER_VALVE_HOPPER_2_UNIT_02"."DATA STANDARD".FEEDBACK_OFF,
                           iPOWDER_FLOW_ON := "DB22133_POWDER_FLOW_HOPPER_2_UNIT_02".oPOWDER_FLOW_ON,
                           MOTOR_STIRRER_SETPOINT := "DB22532_STIRRER_CONTROL_HOPPER_2_UNIT_02"."PROGRAM _SETPOINT _VELOCITY",
                           PRESSURE_SETPOINT := "DB22533_PRESSURE_CONTROL_HOPPER_2_UNIT_02".PRESSURE_SETPOINT_AUTO,
                           oEXCEEDED_TIME_ALARM => "DB426_ALARMS_WARNINGS".CLADDING_HOPPERS."717480",
                           oOUT_OF_RANGE_ALARM => "DB426_ALARMS_WARNINGS".CLADDING_HOPPERS."717481",
                           oLOST_CONDITIONS => "DB426_ALARMS_WARNINGS".CLADDING_HOPPERS."717482");
END_REGION

REGION Network 14: CALL FB22702 LOAD FEEDER SEQUENCE WEIGHT UNIT 02 HOPPER 2
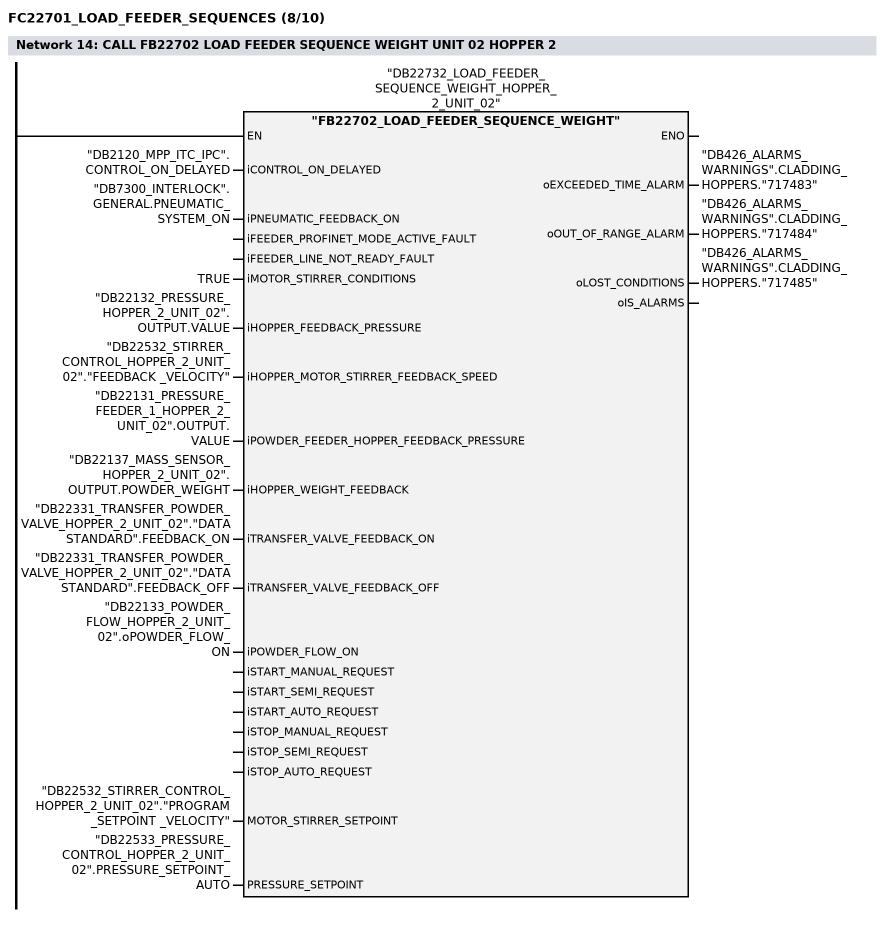
   RUNG wire#powerrail
      "DB22732_LOAD_FEEDER_SEQUENCE_WEIGHT_HOPPER_2_UNIT_02"(iCONTROL_ON_DELAYED := "DB2120_MPP_ITC_IPC".CONTROL_ON_DELAYED, iPNEUMATIC_FEEDBACK_ON := "DB7300_INTERLOCK".GENERAL.PNEUMATIC_SYSTEM_ON, iFEEDER_PROFINET_MODE_ACTIVE_FAULT :=, iFEEDER_LINE_NOT_READY_FAULT :=, iMOTOR_STIRRER_CONDITIONS := TRUE, iHOPPER_FEEDBACK_PRESSURE := "DB22132_PRESSURE_HOPPER_2_UNIT_02".OUTPUT.VALUE, iHOPPER_MOTOR_STIRRER_FEEDBACK_SPEED := "DB22532_STIRRER_CONTROL_HOPPER_2_UNIT_02"."FEEDBACK _VELOCITY", iPOWDER_FEEDER_HOPPER_FEEDBACK_PRESSURE := "DB22131_PRESSURE_FEEDER_1_HOPPER_2_UNIT_02".OUTPUT.VALUE, iHOPPER_WEIGHT_FEEDBACK := "DB22137_MASS_SENSOR_HOPPER_2_UNIT_02".OUTPUT.POWDER_WEIGHT, iTRANSFER_VALVE_FEEDBACK_ON := "DB22331_TRANSFER_POWDER_VALVE_HOPPER_2_UNIT_02"."DATA STANDARD".FEEDBACK_ON, iTRANSFER_VALVE_FEEDBACK_OFF := "DB22331_TRANSFER_POWDER_VALVE_HOPPER_2_UNIT_02"."DATA STANDARD".FEEDBACK_OFF, iPOWDER_FLOW_ON := "DB22133_POWDER_FLOW_HOPPER_2_UNIT_02".oPOWDER_FLOW_ON, iSTART_MANUAL_REQUEST :=, iSTART_SEMI_REQUEST :=, iSTART_AUTO_REQUEST :=, iSTOP_MANUAL_REQUEST :=, iSTOP_SEMI_REQUEST :=, iSTOP_AUTO_REQUEST :=, MOTOR_STIRRER_SETPOINT := "DB22532_STIRRER_CONTROL_HOPPER_2_UNIT_02"."PROGRAM _SETPOINT _VELOCITY", PRESSURE_SETPOINT := "DB22533_PRESSURE_CONTROL_HOPPER_2_UNIT_02".PRESSURE_SETPOINT_AUTO, oEXCEEDED_TIME_ALARM => "DB426_ALARMS_WARNINGS".CLADDING_HOPPERS."717483", oOUT_OF_RANGE_ALARM => "DB426_ALARMS_WARNINGS".CLADDING_HOPPERS."717484", oLOST_CONDITIONS => "DB426_ALARMS_WARNINGS".CLADDING_HOPPERS."717485", oIS_ALARMS =>)
   END_RUNG
   // the same network as SCL:
   "DB22732_LOAD_FEEDER_SEQUENCE_WEIGHT_HOPPER_2_UNIT_02"(iCONTROL_ON_DELAYED := "DB2120_MPP_ITC_IPC".CONTROL_ON_DELAYED,   // "FB22702_LOAD_FEEDER_SEQUENCE_WEIGHT"
                           iPNEUMATIC_FEEDBACK_ON := "DB7300_INTERLOCK".GENERAL.PNEUMATIC_SYSTEM_ON,
                           iMOTOR_STIRRER_CONDITIONS := TRUE,
                           iHOPPER_FEEDBACK_PRESSURE := "DB22132_PRESSURE_HOPPER_2_UNIT_02".OUTPUT.VALUE,
                           iHOPPER_MOTOR_STIRRER_FEEDBACK_SPEED := "DB22532_STIRRER_CONTROL_HOPPER_2_UNIT_02"."FEEDBACK _VELOCITY",
                           iPOWDER_FEEDER_HOPPER_FEEDBACK_PRESSURE := "DB22131_PRESSURE_FEEDER_1_HOPPER_2_UNIT_02".OUTPUT.VALUE,
                           iHOPPER_WEIGHT_FEEDBACK := "DB22137_MASS_SENSOR_HOPPER_2_UNIT_02".OUTPUT.POWDER_WEIGHT,
                           iTRANSFER_VALVE_FEEDBACK_ON := "DB22331_TRANSFER_POWDER_VALVE_HOPPER_2_UNIT_02"."DATA STANDARD".FEEDBACK_ON,
                           iTRANSFER_VALVE_FEEDBACK_OFF := "DB22331_TRANSFER_POWDER_VALVE_HOPPER_2_UNIT_02"."DATA STANDARD".FEEDBACK_OFF,
                           iPOWDER_FLOW_ON := "DB22133_POWDER_FLOW_HOPPER_2_UNIT_02".oPOWDER_FLOW_ON,
                           MOTOR_STIRRER_SETPOINT := "DB22532_STIRRER_CONTROL_HOPPER_2_UNIT_02"."PROGRAM _SETPOINT _VELOCITY",
                           PRESSURE_SETPOINT := "DB22533_PRESSURE_CONTROL_HOPPER_2_UNIT_02".PRESSURE_SETPOINT_AUTO,
                           oEXCEEDED_TIME_ALARM => "DB426_ALARMS_WARNINGS".CLADDING_HOPPERS."717483",
                           oOUT_OF_RANGE_ALARM => "DB426_ALARMS_WARNINGS".CLADDING_HOPPERS."717484",
                           oLOST_CONDITIONS => "DB426_ALARMS_WARNINGS".CLADDING_HOPPERS."717485");
END_REGION

REGION Network 15: /////_HOPPER_3_SEQUENCES_/////
END_REGION

REGION Network 16: CALL FB22701 LOAD FEEDER SEQUENCE TIME UNIT 02 HOPPER 3
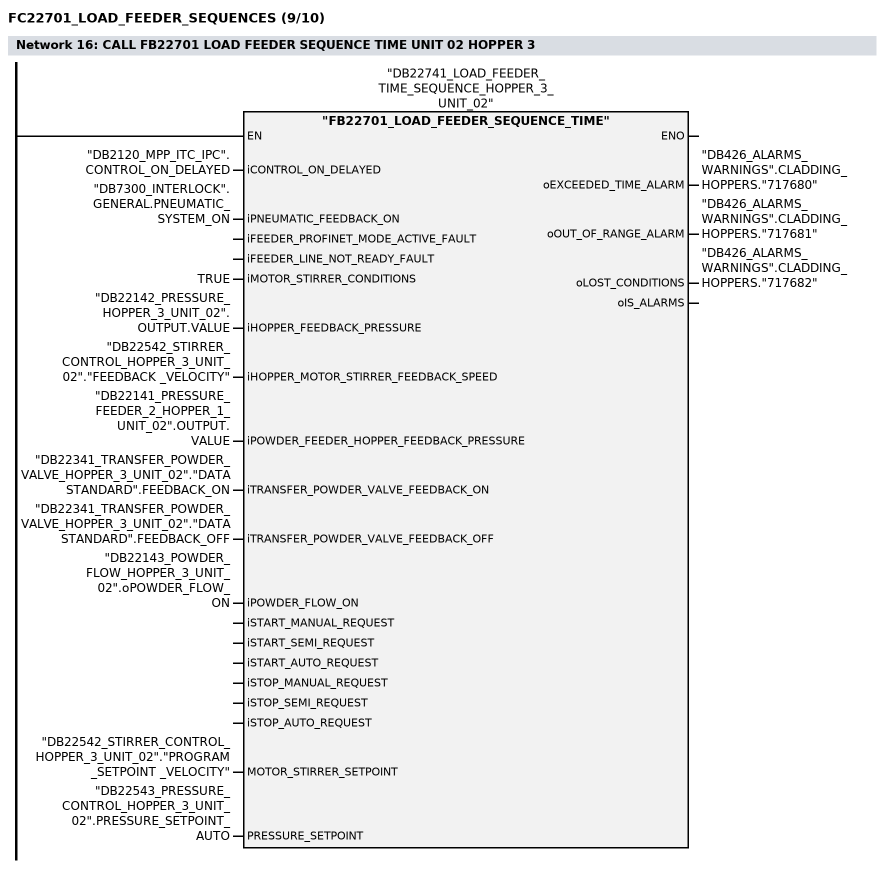
   RUNG wire#powerrail
      "DB22741_LOAD_FEEDER_TIME_SEQUENCE_HOPPER_3_UNIT_02"(iCONTROL_ON_DELAYED := "DB2120_MPP_ITC_IPC".CONTROL_ON_DELAYED, iPNEUMATIC_FEEDBACK_ON := "DB7300_INTERLOCK".GENERAL.PNEUMATIC_SYSTEM_ON, iFEEDER_PROFINET_MODE_ACTIVE_FAULT :=, iFEEDER_LINE_NOT_READY_FAULT :=, iMOTOR_STIRRER_CONDITIONS := TRUE, iHOPPER_FEEDBACK_PRESSURE := "DB22142_PRESSURE_HOPPER_3_UNIT_02".OUTPUT.VALUE, iHOPPER_MOTOR_STIRRER_FEEDBACK_SPEED := "DB22542_STIRRER_CONTROL_HOPPER_3_UNIT_02"."FEEDBACK _VELOCITY", iPOWDER_FEEDER_HOPPER_FEEDBACK_PRESSURE := "DB22141_PRESSURE_FEEDER_2_HOPPER_1_UNIT_02".OUTPUT.VALUE, iTRANSFER_POWDER_VALVE_FEEDBACK_ON := "DB22341_TRANSFER_POWDER_VALVE_HOPPER_3_UNIT_02"."DATA STANDARD".FEEDBACK_ON, iTRANSFER_POWDER_VALVE_FEEDBACK_OFF := "DB22341_TRANSFER_POWDER_VALVE_HOPPER_3_UNIT_02"."DATA STANDARD".FEEDBACK_OFF, iPOWDER_FLOW_ON := "DB22143_POWDER_FLOW_HOPPER_3_UNIT_02".oPOWDER_FLOW_ON, iSTART_MANUAL_REQUEST :=, iSTART_SEMI_REQUEST :=, iSTART_AUTO_REQUEST :=, iSTOP_MANUAL_REQUEST :=, iSTOP_SEMI_REQUEST :=, iSTOP_AUTO_REQUEST :=, MOTOR_STIRRER_SETPOINT := "DB22542_STIRRER_CONTROL_HOPPER_3_UNIT_02"."PROGRAM _SETPOINT _VELOCITY", PRESSURE_SETPOINT := "DB22543_PRESSURE_CONTROL_HOPPER_3_UNIT_02".PRESSURE_SETPOINT_AUTO, oEXCEEDED_TIME_ALARM => "DB426_ALARMS_WARNINGS".CLADDING_HOPPERS."717680", oOUT_OF_RANGE_ALARM => "DB426_ALARMS_WARNINGS".CLADDING_HOPPERS."717681", oLOST_CONDITIONS => "DB426_ALARMS_WARNINGS".CLADDING_HOPPERS."717682", oIS_ALARMS =>)
   END_RUNG
   // the same network as SCL:
   "DB22741_LOAD_FEEDER_TIME_SEQUENCE_HOPPER_3_UNIT_02"(iCONTROL_ON_DELAYED := "DB2120_MPP_ITC_IPC".CONTROL_ON_DELAYED,   // "FB22701_LOAD_FEEDER_SEQUENCE_TIME"
                           iPNEUMATIC_FEEDBACK_ON := "DB7300_INTERLOCK".GENERAL.PNEUMATIC_SYSTEM_ON,
                           iMOTOR_STIRRER_CONDITIONS := TRUE,
                           iHOPPER_FEEDBACK_PRESSURE := "DB22142_PRESSURE_HOPPER_3_UNIT_02".OUTPUT.VALUE,
                           iHOPPER_MOTOR_STIRRER_FEEDBACK_SPEED := "DB22542_STIRRER_CONTROL_HOPPER_3_UNIT_02"."FEEDBACK _VELOCITY",
                           iPOWDER_FEEDER_HOPPER_FEEDBACK_PRESSURE := "DB22141_PRESSURE_FEEDER_2_HOPPER_1_UNIT_02".OUTPUT.VALUE,
                           iTRANSFER_POWDER_VALVE_FEEDBACK_ON := "DB22341_TRANSFER_POWDER_VALVE_HOPPER_3_UNIT_02"."DATA STANDARD".FEEDBACK_ON,
                           iTRANSFER_POWDER_VALVE_FEEDBACK_OFF := "DB22341_TRANSFER_POWDER_VALVE_HOPPER_3_UNIT_02"."DATA STANDARD".FEEDBACK_OFF,
                           iPOWDER_FLOW_ON := "DB22143_POWDER_FLOW_HOPPER_3_UNIT_02".oPOWDER_FLOW_ON,
                           MOTOR_STIRRER_SETPOINT := "DB22542_STIRRER_CONTROL_HOPPER_3_UNIT_02"."PROGRAM _SETPOINT _VELOCITY",
                           PRESSURE_SETPOINT := "DB22543_PRESSURE_CONTROL_HOPPER_3_UNIT_02".PRESSURE_SETPOINT_AUTO,
                           oEXCEEDED_TIME_ALARM => "DB426_ALARMS_WARNINGS".CLADDING_HOPPERS."717680",
                           oOUT_OF_RANGE_ALARM => "DB426_ALARMS_WARNINGS".CLADDING_HOPPERS."717681",
                           oLOST_CONDITIONS => "DB426_ALARMS_WARNINGS".CLADDING_HOPPERS."717682");
END_REGION

REGION Network 17: CALL FB22702 LOAD FEEDER SEQUENCE WEIGHT UNIT 02 HOPPER 3
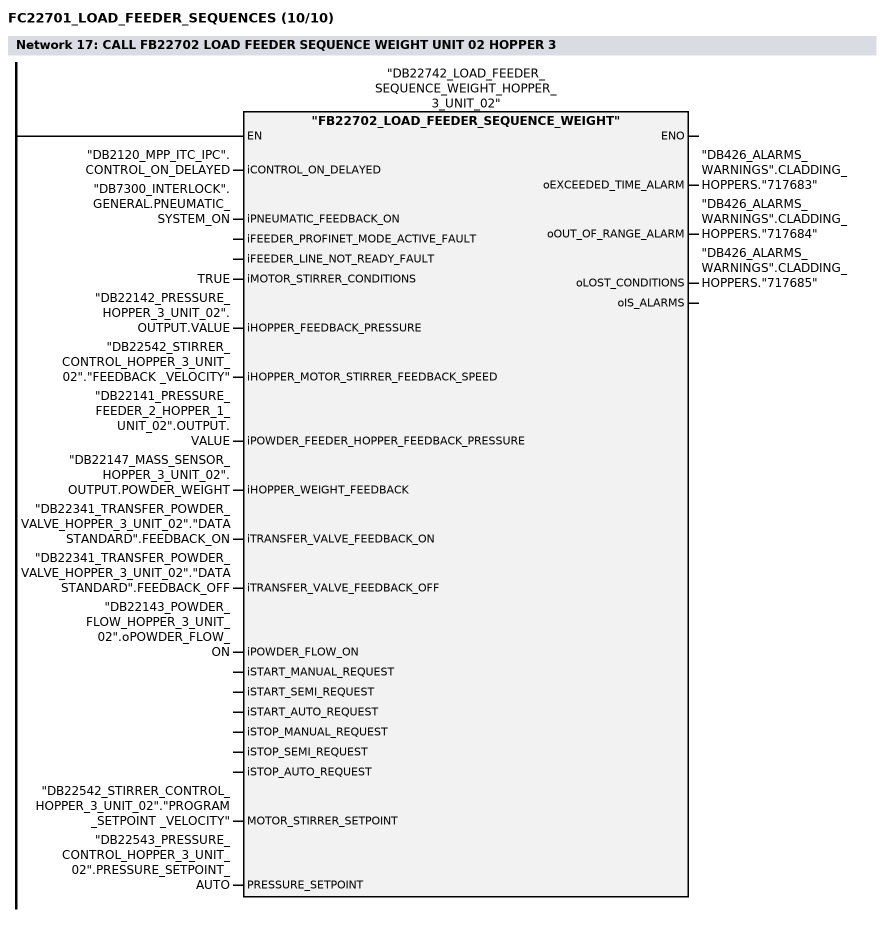
   RUNG wire#powerrail
      "DB22742_LOAD_FEEDER_SEQUENCE_WEIGHT_HOPPER_3_UNIT_02"(iCONTROL_ON_DELAYED := "DB2120_MPP_ITC_IPC".CONTROL_ON_DELAYED, iPNEUMATIC_FEEDBACK_ON := "DB7300_INTERLOCK".GENERAL.PNEUMATIC_SYSTEM_ON, iFEEDER_PROFINET_MODE_ACTIVE_FAULT :=, iFEEDER_LINE_NOT_READY_FAULT :=, iMOTOR_STIRRER_CONDITIONS := TRUE, iHOPPER_FEEDBACK_PRESSURE := "DB22142_PRESSURE_HOPPER_3_UNIT_02".OUTPUT.VALUE, iHOPPER_MOTOR_STIRRER_FEEDBACK_SPEED := "DB22542_STIRRER_CONTROL_HOPPER_3_UNIT_02"."FEEDBACK _VELOCITY", iPOWDER_FEEDER_HOPPER_FEEDBACK_PRESSURE := "DB22141_PRESSURE_FEEDER_2_HOPPER_1_UNIT_02".OUTPUT.VALUE, iHOPPER_WEIGHT_FEEDBACK := "DB22147_MASS_SENSOR_HOPPER_3_UNIT_02".OUTPUT.POWDER_WEIGHT, iTRANSFER_VALVE_FEEDBACK_ON := "DB22341_TRANSFER_POWDER_VALVE_HOPPER_3_UNIT_02"."DATA STANDARD".FEEDBACK_ON, iTRANSFER_VALVE_FEEDBACK_OFF := "DB22341_TRANSFER_POWDER_VALVE_HOPPER_3_UNIT_02"."DATA STANDARD".FEEDBACK_OFF, iPOWDER_FLOW_ON := "DB22143_POWDER_FLOW_HOPPER_3_UNIT_02".oPOWDER_FLOW_ON, iSTART_MANUAL_REQUEST :=, iSTART_SEMI_REQUEST :=, iSTART_AUTO_REQUEST :=, iSTOP_MANUAL_REQUEST :=, iSTOP_SEMI_REQUEST :=, iSTOP_AUTO_REQUEST :=, MOTOR_STIRRER_SETPOINT := "DB22542_STIRRER_CONTROL_HOPPER_3_UNIT_02"."PROGRAM _SETPOINT _VELOCITY", PRESSURE_SETPOINT := "DB22543_PRESSURE_CONTROL_HOPPER_3_UNIT_02".PRESSURE_SETPOINT_AUTO, oEXCEEDED_TIME_ALARM => "DB426_ALARMS_WARNINGS".CLADDING_HOPPERS."717683", oOUT_OF_RANGE_ALARM => "DB426_ALARMS_WARNINGS".CLADDING_HOPPERS."717684", oLOST_CONDITIONS => "DB426_ALARMS_WARNINGS".CLADDING_HOPPERS."717685", oIS_ALARMS =>)
   END_RUNG
   // the same network as SCL:
   "DB22742_LOAD_FEEDER_SEQUENCE_WEIGHT_HOPPER_3_UNIT_02"(iCONTROL_ON_DELAYED := "DB2120_MPP_ITC_IPC".CONTROL_ON_DELAYED,   // "FB22702_LOAD_FEEDER_SEQUENCE_WEIGHT"
                           iPNEUMATIC_FEEDBACK_ON := "DB7300_INTERLOCK".GENERAL.PNEUMATIC_SYSTEM_ON,
                           iMOTOR_STIRRER_CONDITIONS := TRUE,
                           iHOPPER_FEEDBACK_PRESSURE := "DB22142_PRESSURE_HOPPER_3_UNIT_02".OUTPUT.VALUE,
                           iHOPPER_MOTOR_STIRRER_FEEDBACK_SPEED := "DB22542_STIRRER_CONTROL_HOPPER_3_UNIT_02"."FEEDBACK _VELOCITY",
                           iPOWDER_FEEDER_HOPPER_FEEDBACK_PRESSURE := "DB22141_PRESSURE_FEEDER_2_HOPPER_1_UNIT_02".OUTPUT.VALUE,
                           iHOPPER_WEIGHT_FEEDBACK := "DB22147_MASS_SENSOR_HOPPER_3_UNIT_02".OUTPUT.POWDER_WEIGHT,
                           iTRANSFER_VALVE_FEEDBACK_ON := "DB22341_TRANSFER_POWDER_VALVE_HOPPER_3_UNIT_02"."DATA STANDARD".FEEDBACK_ON,
                           iTRANSFER_VALVE_FEEDBACK_OFF := "DB22341_TRANSFER_POWDER_VALVE_HOPPER_3_UNIT_02"."DATA STANDARD".FEEDBACK_OFF,
                           iPOWDER_FLOW_ON := "DB22143_POWDER_FLOW_HOPPER_3_UNIT_02".oPOWDER_FLOW_ON,
                           MOTOR_STIRRER_SETPOINT := "DB22542_STIRRER_CONTROL_HOPPER_3_UNIT_02"."PROGRAM _SETPOINT _VELOCITY",
                           PRESSURE_SETPOINT := "DB22543_PRESSURE_CONTROL_HOPPER_3_UNIT_02".PRESSURE_SETPOINT_AUTO,
                           oEXCEEDED_TIME_ALARM => "DB426_ALARMS_WARNINGS".CLADDING_HOPPERS."717683",
                           oOUT_OF_RANGE_ALARM => "DB426_ALARMS_WARNINGS".CLADDING_HOPPERS."717684",
                           oLOST_CONDITIONS => "DB426_ALARMS_WARNINGS".CLADDING_HOPPERS."717685");
END_REGION
END_FUNCTION
